PROGRAM P4_00_MAIN
VAR
END_VAR

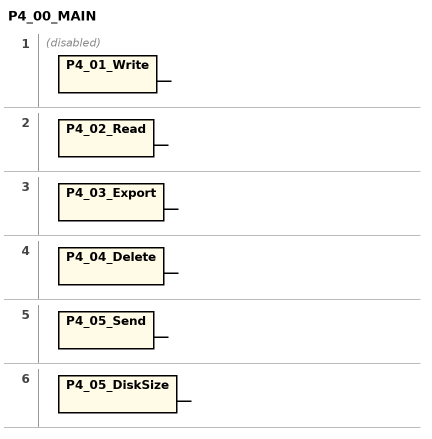
// NETWORK 1 (disabled)
// P4_01_Write();

// NETWORK 2
P4_02_Read();

// NETWORK 3
P4_03_Export();

// NETWORK 4
P4_04_Delete();

// NETWORK 5
P4_05_Send();

// NETWORK 6
P4_05_DiskSize();

END_PROGRAM

(* stored: Version 1.1.0.1
   POU P4_00_MAIN: Id {d511578b-b7de-42e9-bf03-fc06d50e5046}, SpecialFunc None *)
